FUNCTION_BLOCK FB_MoveRequest_Test EXTENDS FB_TestSuite
VAR
        stMotionEpicsItf :  ST_MotionEpicsInterface;
END_VAR

GivenMoveCmdCheckDriveInputThenCheckRequestAndEpicsStatus();

METHOD GivenEpicsExecuteCheckDriveInputThenCheckRequestAndEpicsStatus
VAR_INPUT
END_VAR
END_METHOD

METHOD GivenHomeCmdCheckDriveInputThenCheckRequestAndEpicsStatus
VAR_INST
    fbMoveRequest : FB_MoveRequest(stMotionEpicsItf:=stMotionEpicsItf);
END_VAR
END_METHOD

METHOD GivenMoveCmdCheckDriveInputThenCheckRequestAndEpicsStatus
VAR
    fbMoveRequest : FB_MoveRequest(stMotionEpicsItf:=stMotionEpicsItf);
    eExpectedMoveMode : INT := E_EpicsMotorCmd.MOVE_ABSOLUTE;
    eActualMoveMode : INT;
END_VAR
TEST(__POUNAME());
fbMoveRequest.MotionRequest(	HomeCmd:=FALSE,
                                MoveCmd:=TRUE,
                                HomeMode:=E_EpicsHomeCmd.NONE,
                                EnableMode:=E_StageEnableMode.DURING_MOTION,
                                EnableDone:=TRUE,
                                MoveOk:=TRUE,
                                PowerEnabled:=TRUE);

fbMoveRequest();

AssertTrue(Condition := fbMoveRequest.NewMoveReq,
           Message := 'New request not Registered #1');
AssertTrue(Condition := fbMoveRequest.Execute,
           Message := 'New request not comfirm for execution #2');
AssertTrue(Condition := fbMoveRequest.ExecMove,
           Message := 'New move request will not execute #3');
AssertFalse(Condition := fbMoveRequest.ExecHome,
           Message := 'The request is not a Homing move #4');
eActualMoveMode :=fbMoveRequest.CommandLocal;
AssertEquals ( Expected:=eExpectedMoveMode, Actual:=eActualMoveMode ,
            Message:='New move request motor  Cmd Must be Absolute #5');
TEST_FINISHED();
END_METHOD

END_FUNCTION_BLOCK

(* stored: Version 1.1.0.1
   POU FB_MoveRequest_Test: Id {05d79949-1f03-4557-a858-9a547a52b2be}, SpecialFunc None
   Method GivenEpicsExecuteCheckDriveInputThenCheckRequestAndEpicsStatus: Id {223fd37a-e346-4e63-ae91-95e8242641a5}
   Method GivenHomeCmdCheckDriveInputThenCheckRequestAndEpicsStatus: Id {9e26be9d-db97-4ea1-b419-a0aadd052025}
   Method GivenMoveCmdCheckDriveInputThenCheckRequestAndEpicsStatus: Id {0278f58c-2e71-49f5-9141-f6fec2b3cd3f} *)
